KUKA KRL program: cell_R1.src

&ACCESS RVP
&REL 5
&COMMENT HANDLER on external automatic
DEF cell_R1( )
  ;EXT EXAMPLE1 ( )
  ;EXT EXAMPLE2 ( )
  ;EXT EXAMPLE3 ( )

  ;FOLD INIT
  DECL CHAR DMY[3]
  DMY[]="---"
  ;ENDFOLD (INIT)
  ;FOLD BASISTECH INI
  GLOBAL INTERRUPT DECL 3 WHEN $STOPMESS==TRUE DO IR_STOPM ( )
  INTERRUPT ON 3
  BAS (#INITMOV,0 )
  ;ENDFOLD (BASISTECH INI)
  ;FOLD CHECK HOME
  $H_POS=XHOME
  IF CHECK_HOME==TRUE THEN
    P00 (#CHK_HOME,#PGNO_GET,DMY[],0 ) ;Testing Home-Position
  ENDIF
  ;ENDFOLD (CHECK HOME)
  ;FOLD PTP HOME  Vel= 100 % DEFAULT;%{PE}%MKUKATPBASIS,%CMOVE,%VPTP,%P 1:PTP, 2:HOME, 3:, 5:100, 7:DEFAULT
  $H_POS=XHOME
  PDAT_ACT=PDEFAULT
  BAS (#PTP_DAT )
  FDAT_ACT=FHOME
  BAS (#FRAMES )
  BAS (#VEL_PTP,100 )
  PTP  XHOME
  ;ENDFOLD
  ;FOLD AUTOEXT INI
  P00 (#INIT_EXT,#PGNO_GET,DMY[],0 ) ; Initialize extern mode
  ;ENDFOLD (AUTOEXT INI)
  LOOP
    P00 (#EXT_PGNO,#PGNO_GET,DMY[],0 )
    SWITCH  PGNO ; Select with Programnumber

    CASE 1 ;PROGRAM DEPALETYZACJI
      P00 (#EXT_PGNO,#PGNO_ACKN,DMY[],0 ) ; Reset Progr.No.-Request

      offline_R1_toolactpos()

    CASE 10 ; PROGRAM SERWISOWY
      P00 (#EXT_PGNO,#PGNO_ACKN,DMY[],0 ) ; Reset Progr.No.-Request

      SERWIS()

    DEFAULT
      P00 (#EXT_PGNO,#PGNO_FAULT,DMY[],0 )
    ENDSWITCH
  ENDLOOP
END
